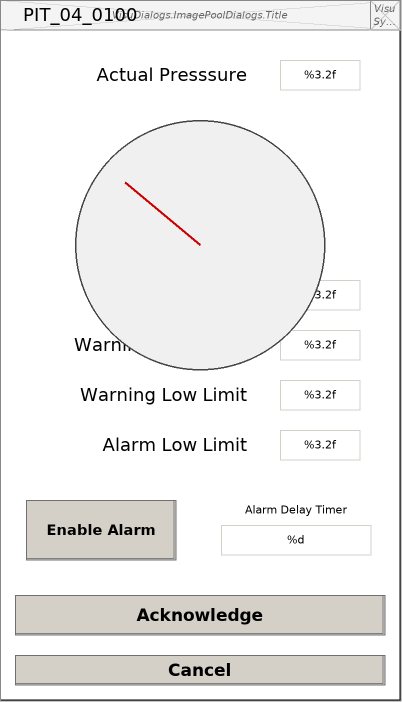
VISUALIZATION visuPITDiag  // 402x702
    Rectangle (0,0 400x700)
    Textfield (280,280 80x30), "%3.2f"
    Button (26,500 150x60), "Enable Alarm"
        toggle progHSVCntrl.HSV_04_0100.EnableAlarm
    Textfield (221,525 150x30), "%d"
    Label (221,495 150x30), "Alarm Delay Timer"
    Image (0,0 400x30), image: VisuDialogs.ImagePoolDialogs.Title
    Group (370,0 30x30)
        RoundedRectangle (0,0 30x30)
        Image (0,0 30x30), image: VisuSymbols.Symbols.Wrong
    Button (15,655 370x30), "Cancel"
    Label (20,0 210x30), "PIT_04_0100"
    Label (0,280 250x30), "Alarm High Limit"
    Label (0,330 250x30), "Warning High Limit"
    Label (0,380 250x30), "Warning Low Limit"
    Label (0,430 250x30), "Alarm Low Limit"
    Textfield (280,330 80x30), "%3.2f"
    Textfield (280,380 80x30), "%3.2f"
    Textfield (280,430 80x30), "%3.2f"
    Button (15,595 370x40), "Acknowledge"
    Textfield (280,60 80x30), "%3.2f"
    Label (0,60 250x30), "Actual Presssure"
    Meter180 (75,120 250x250), style: Meter-Meter180-Gray, scale format: %.1f, scale 0..100
END_VISUALIZATION

(* stored: Version 1.1.0.1, ProductVersion 3.1.4022.17
   Visu visuPITDiag: Id {5b2871b6-d1d3-49ef-932b-a1f3e5234741} *)
